(* IEC 61131-3 sources: RL_MAR/experiments/comparison/autoplc/results/gpt-4o_20260511_211137/med_52, 1 file *)

(* ---- med_52_1.st ---- *)
FUNCTION_BLOCK TrafficManagementSystem
    VAR_INPUT
        VehicleCount1 : INT;
        VehicleCount2 : INT;
        VehicleCount3 : INT;
        VehicleCount4 : INT;
    END_VAR

    VAR_OUTPUT
        TrafficLight1 : BOOL;
        TrafficLight2 : BOOL;
        TrafficLight3 : BOOL;
        TrafficLight4 : BOOL;
    END_VAR

    VAR
        // Internal variables can be declared here if needed
    END_VAR

    // Initialize the traffic lights with default states
    TrafficLight1 := FALSE; // Red
    TrafficLight2 := TRUE;  // Green
    TrafficLight3 := FALSE; // Red
    TrafficLight4 := TRUE;  // Green

    // Continuously monitor and update traffic light states based on vehicle counts
    IF VehicleCount1 > VehicleCount2 THEN
        TrafficLight1 := TRUE;  // Green
        TrafficLight2 := FALSE; // Red
    ELSE
        TrafficLight1 := FALSE; // Red
        TrafficLight2 := TRUE;  // Green
    END_IF

    IF VehicleCount3 > VehicleCount4 THEN
        TrafficLight3 := TRUE;  // Green
        TrafficLight4 := FALSE; // Red
    ELSE
        TrafficLight3 := FALSE; // Red
        TrafficLight4 := TRUE;  // Green
    END_IF
END_FUNCTION_BLOCK
